// Mitsubishi GX Works2 project: 평가 프로젝트_김채린   PLC: Q02/Q02H

PROGRAM MAIN
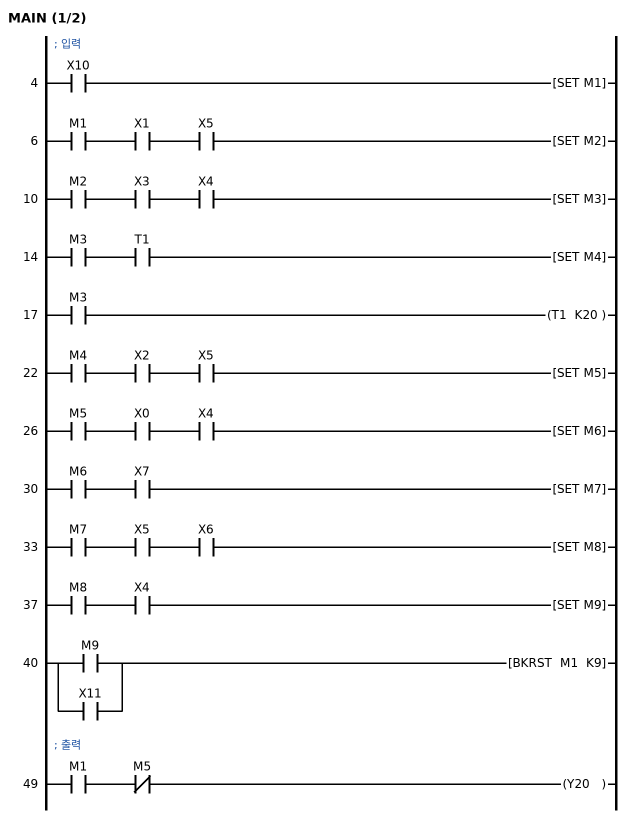
; 입력
4     LD      X10
      SET     M1
6     LD      M1
      AND     X1
      AND     X5
      SET     M2
10    LD      M2
      AND     X3
      AND     X4
      SET     M3
14    LD      M3
      AND     T1
      SET     M4
17    LD      M3
      OUT     T1 K20
22    LD      M4
      AND     X2
      AND     X5
      SET     M5
26    LD      M5
      AND     X0
      AND     X4
      SET     M6
30    LD      M6
      AND     X7
      SET     M7
33    LD      M7
      AND     X5
      AND     X6
      SET     M8
37    LD      M8
      AND     X4
      SET     M9
40    LD      M9
      OR      X11
      BKRST   M1 K9
; 출력
49    LD      M1
      ANI     M5
      OUT     Y20
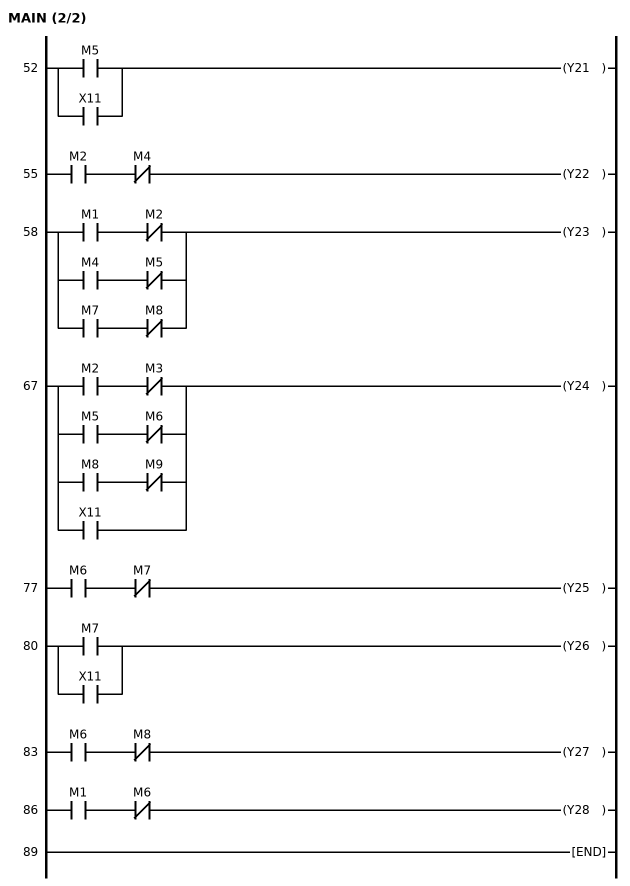
52    LD      M5
      OR      X11
      OUT     Y21
55    LD      M2
      ANI     M4
      OUT     Y22
58    LD      M1
      ANI     M2
      LD      M4
      ANI     M5
      ORB
      LD      M7
      ANI     M8
      ORB
      OUT     Y23
67    LD      M2
      ANI     M3
      LD      M5
      ANI     M6
      ORB
      LD      M8
      ANI     M9
      ORB
      OR      X11
      OUT     Y24
77    LD      M6
      ANI     M7
      OUT     Y25
80    LD      M7
      OR      X11
      OUT     Y26
83    LD      M6
      ANI     M8
      OUT     Y27
86    LD      M1
      ANI     M6
      OUT     Y28
89    END
END_PROGRAM

PROGRAM HMI
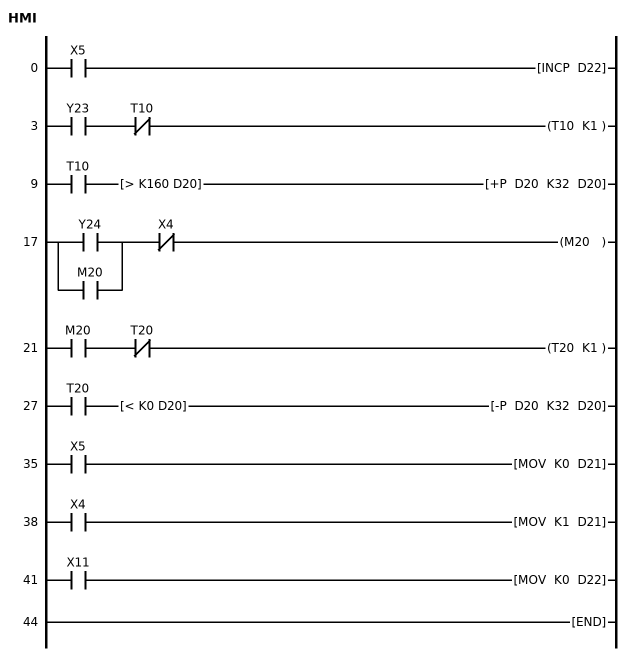
0     LD      X5
      INCP    D22
3     LD      Y23
      ANI     T10
      OUT     T10 K1
9     LD      T10
      AND>    K160 D20
      +P      D20 K32 D20
17    LD      Y24
      OR      M20
      ANI     X4
      OUT     M20
21    LD      M20
      ANI     T20
      OUT     T20 K1
27    LD      T20
      AND<    K0 D20
      -P      D20 K32 D20
35    LD      X5
      MOV     K0 D21
38    LD      X4
      MOV     K1 D21
41    LD      X11
      MOV     K0 D22
44    END
END_PROGRAM
